// TIA Portal V20 export
// export: Created 2026-07-10T11:12:26.991727Z, ExportSetting WithDefaults, DisplayName Totally Integrated Automation Portal, DisplayVersion V20, DisplayName TIA Portal Openness, DisplayVersion V20, DisplayName TIA Portal Version Control Interface, DisplayVersion V20, DisplayName STEP 7 Professional, DisplayVersion V20, DisplayName STEP 7 Safety, DisplayVersion V20, DisplayName WinCC Basic/Comfort/Advanced, DisplayVersion V20, DisplayName WinCC Unified, DisplayVersion V20
DATA_BLOCK "WaterCounter_DB"   // DB2
VERSION : 0.1
// stored: AutoNumber true, DBAccessibleFromOPCUA true, InstanceOfName WaterCounter, InstanceOfType FB
"WaterCounter"
   // VAR
   //    WaterCounter_InWater : "FlowCounter";
   //    WaterCounter_OutWater : "FlowCounter";
   //    DelayTON { S7_SetPoint := 'True'} : TON_TIME;
   //    ChlorCounter_1 { S7_SetPoint := 'True'} : "FlowCounter";
   //    ChlorCounter_2 { S7_SetPoint := 'True'} : "FlowCounter";
   // END_VAR
BEGIN
END_DATA_BLOCK
